# EPICS substitutions: iocs/MC06/MCApp/Db-orig/SAI_DigitalChannels.substitutions
file /opt/epics/modules/SAI/db/SAI_DigitalChannels.template {
pattern {	P,		R,		SCAN, 		ASYNPORT}
        { 	"XF:06BM-OP",		"{MC:01}",	"1 second",	"pmac"}
}

#EOF
